(* Base of Control Primitives. Inheriting FBs must implement the type-specific "ExecuteInternal" method. *)
FUNCTION_BLOCK ABSTRACT ControlPrimitiveBase EXTENDS BehaviorBase
VAR
	m_timeout: TIME;
	
	m_internalRes: BOOL;
	m_pre: IExpression;
	m_post: IExpression;
	
	// store the conditions as string for access via OPC UA + easier debugging
	{attribute 'OPC.UA.DA' := '1'}
	{attribute 'OPC.UA.DA.Access' := '1'}
	m_preStr: STRING(256);
	{attribute 'OPC.UA.DA' := '1'}
	{attribute 'OPC.UA.DA.Access' := '1'}
	m_postStr: STRING(256);
	
	m_st: POINTER TO StateTracker;
	m_pm: POINTER TO ProcessManager;
	
	m_tonTimeout: TON;
	
	m_didAbort: BOOL;
END_VAR

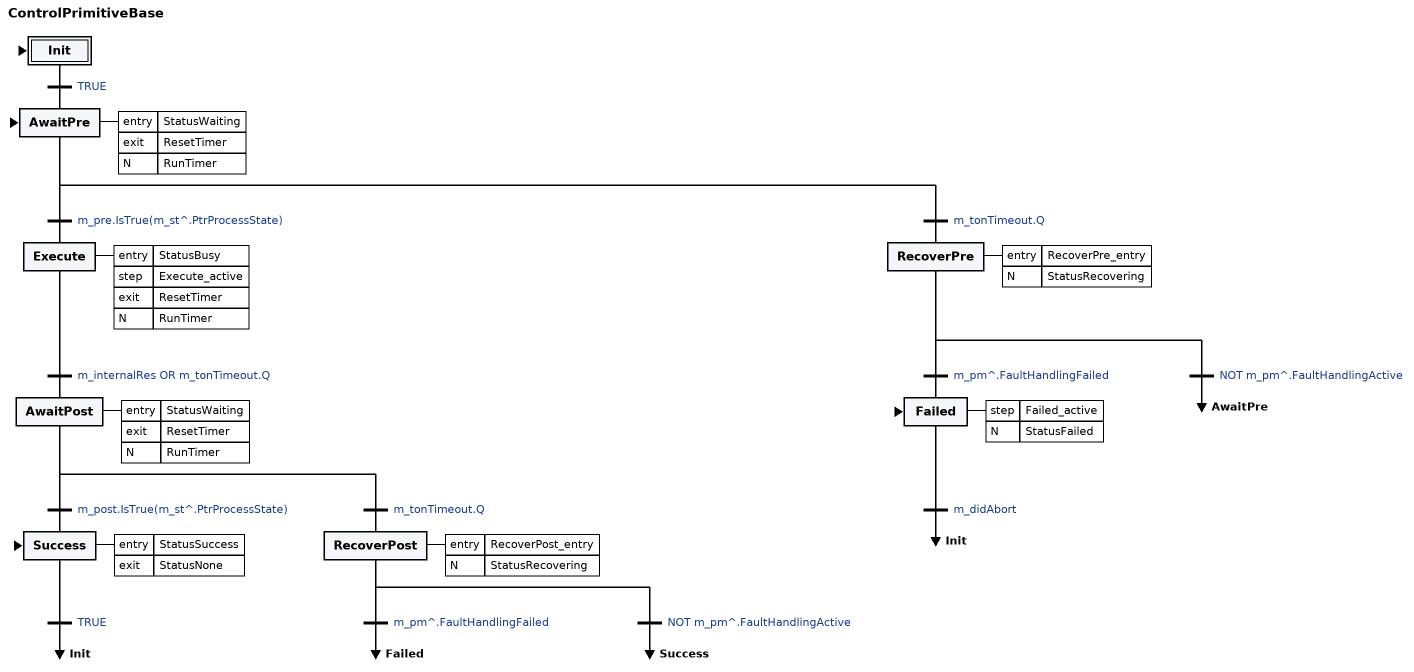
INITIAL_STEP Init:
END_STEP
TRANSITION FROM Init TO AwaitPre
    := TRUE;
END_TRANSITION
STEP AwaitPre:
    StatusWaiting(P1);  // entry action
    ResetTimer(P0);  // exit action
    RunTimer(N);
END_STEP
TRANSITION FROM AwaitPre TO Execute
    := m_pre.IsTrue(m_st^.PtrProcessState);
END_TRANSITION
STEP Execute:
    StatusBusy(P1);  // entry action
    Execute_active(N);  // step action
    ResetTimer(P0);  // exit action
    RunTimer(N);
END_STEP
TRANSITION FROM Execute TO AwaitPost
    := m_internalRes OR m_tonTimeout.Q;
END_TRANSITION
STEP AwaitPost:
    StatusWaiting(P1);  // entry action
    ResetTimer(P0);  // exit action
    RunTimer(N);
END_STEP
TRANSITION FROM AwaitPost TO Success
    := m_post.IsTrue(m_st^.PtrProcessState);
END_TRANSITION
STEP Success:
    StatusSuccess(P1);  // entry action
    StatusNone(P0);  // exit action
END_STEP
TRANSITION FROM Success TO Init
    := TRUE;
END_TRANSITION
TRANSITION FROM AwaitPost TO RecoverPost
    := m_tonTimeout.Q;
END_TRANSITION
STEP RecoverPost:
    RecoverPost_entry(P1);  // entry action
    StatusRecovering(N);
END_STEP
TRANSITION FROM RecoverPost TO Failed
    := m_pm^.FaultHandlingFailed;
END_TRANSITION
TRANSITION FROM RecoverPost TO Success
    := NOT m_pm^.FaultHandlingActive;
END_TRANSITION
TRANSITION FROM AwaitPre TO RecoverPre
    := m_tonTimeout.Q;
END_TRANSITION
STEP RecoverPre:
    RecoverPre_entry(P1);  // entry action
    StatusRecovering(N);
END_STEP
TRANSITION FROM RecoverPre TO Failed
    := m_pm^.FaultHandlingFailed;
END_TRANSITION
STEP Failed:
    Failed_active(N);  // step action
    StatusFailed(N);
END_STEP
TRANSITION FROM Failed TO Init
    := m_didAbort;
END_TRANSITION
TRANSITION FROM RecoverPre TO AwaitPre
    := NOT m_pm^.FaultHandlingActive;
END_TRANSITION

METHOD ABSTRACT Abort : BOOL
VAR_INPUT
END_VAR
END_METHOD

ACTION Execute_active:
IF NOT m_internalRes THEN
	m_internalRes := ExecuteInternal(i_params);
END_IF
END_ACTION

(* Execution logic of this Control Primitive. *)
METHOD PROTECTED ABSTRACT ExecuteInternal : BOOL
VAR_INPUT
	i_params: ParameterSet;
END_VAR
END_METHOD

ACTION Failed_active:
m_didAbort := Abort();
END_ACTION

PROPERTY Postcondition : IExpression
GET
Postcondition := m_post;
END_GET
SET
m_post := Postcondition;
m_postStr := Postcondition.ToString();
END_SET
END_PROPERTY

PROPERTY Precondition : IExpression
GET
Precondition := m_pre;
END_GET
SET
m_pre := Precondition;
m_preStr := Precondition.ToString();
END_SET
END_PROPERTY

METHOD ProvideServices : BOOL
VAR_INPUT
	i_ptrProcessManager: POINTER TO ProcessManager;
	i_ptrStateTracker: POINTER TO StateTracker;
END_VAR
m_pm := i_ptrProcessManager;
m_st := i_ptrStateTracker;
END_METHOD

ACTION RecoverPost_entry:
m_pm^.RequestRecovery(m_post, CONCAT('Primitive ', TO_STRING(m_id)));
END_ACTION

ACTION RecoverPre_entry:
m_pm^.RequestRecovery(m_pre, CONCAT('Primitive ', TO_STRING(m_id)));
END_ACTION

ACTION ResetTimer:
m_tonTimeout(IN := FALSE);
m_internalRes := FALSE;
END_ACTION

ACTION RunTimer:
m_tonTimeout(IN := TRUE, PT := m_timeout);
END_ACTION

ACTION StatusBusy:
o_status := EOperationResult.busy;
END_ACTION

ACTION StatusFailed:
o_status := EOperationResult.failed;
END_ACTION

ACTION StatusNone:
o_status := EOperationResult.none;
END_ACTION

ACTION StatusRecovering:
o_status := EOperationResult.recovering;
END_ACTION

ACTION StatusSuccess:
o_status := EOperationResult.success;
END_ACTION

ACTION StatusWaiting:
o_status := EOperationResult.waiting;
END_ACTION

END_FUNCTION_BLOCK

(* stored: Version 1.1.0.1
   POU ControlPrimitiveBase: Id {b043c000-3860-4c94-89ff-cc224924a18d}, SpecialFunc None
   Folder Actions: Id {26724dad-172e-4616-92eb-ca41c77864ac}
   Method Abort: Id {4a07d954-ae1d-4956-bc45-8d59c82d1704}
   Action Execute_active: Id {9fb5ba26-19e1-44ec-a5f9-5888c01ee93c}
   Method ExecuteInternal: Id {fce5a6e9-06f8-40c9-b9ba-4e816dac0899}
   Action Failed_active: Id {1974abd5-4c2e-4df4-b5a0-dc33db09342d}
   Property Postcondition: Id {5df2da4f-d4c6-4d05-acdb-c45aafebf1b3}
   Get Get: Id {55d31a3d-3632-4345-80eb-060c7da9f01d}
   Set Set: Id {f4d2e9c7-413e-4144-a1f7-8e80e46db4ae}
   Property Precondition: Id {1e22b21e-08a0-47f5-9ed9-8589058c8203}
   Get Get: Id {e7a08402-fcb1-4b06-8f6c-6c760609fa90}
   Set Set: Id {d3b7dde0-f7e1-4ef7-ba6f-e553ea9532c8}
   Method ProvideServices: Id {f6897f65-baaf-4986-a6ac-a5d6167d9047}
   Action RecoverPost_entry: Id {e57d9529-b2bf-49df-a6ce-01ee11eacaad}
   Action RecoverPre_entry: Id {04c43ee0-95f8-4da0-88c4-77db83763ba9}
   Action ResetTimer: Id {8653afe2-8765-4186-b958-fee58caf2875}
   Action RunTimer: Id {c745ff60-9393-40ae-9663-2e01972666c4}
   Action StatusBusy: Id {031f5dbf-ca58-4422-9def-a0c6bcc8d13d}
   Action StatusFailed: Id {105db533-690d-4cc0-b7d8-ebb23e30ea01}
   Action StatusNone: Id {8f54d379-c858-4bf6-a6ee-a04d4aed6393}
   Action StatusRecovering: Id {cbc3c96d-310e-46ef-8c42-48b9d7180f05}
   Action StatusSuccess: Id {11621188-2fdb-4f77-aed9-fa613c6ef03b}
   Action StatusWaiting: Id {7b3faaac-8f94-48d7-909b-0cae464e7905} *)
